FUNCTION VecSum : Vec3
VAR_INPUT
	a : ARRAY[0..3] OF Vec3; 
END_VAR
VAR
	i: INT;
	sum : Vec3;
END_VAR

sum := SetVec3(0, 0, 0);
FOR i := 0 TO 3 DO
	sum := VecAdd(sum, a[i]);
END_FOR
VecSum := sum;

END_FUNCTION

(* stored: Version 1.1.0.1, ProductVersion 3.1.4024.2
   POU VecSum: Id {8bbe2ea5-a582-4b33-aecd-eae4ceee4ebe}, SpecialFunc None *)
